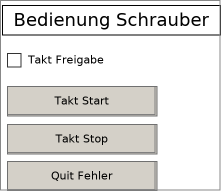
VISUALIZATION Frame_Schrauber_Bedien  // 221x191
VAR_IN_OUT
	bTaktFreigabe	:BOOL;
	bTaktStart		:BOOL;
	bTaktStop		:BOOL;
	bQuitError		:BOOL;
	
END_VAR
    Button (7,124 150x30), "Takt Stop"
        tap bTaktStop
    Button (7,86 150x30), "Takt Start"
        tap bTaktStart
    Checkbox (5,45 150x30), "Takt Freigabe", variable: bTaktFreigabe
    Rectangle (2,5 219x30), "Bedienung Schrauber"
    Button (7,161 150x30), "Quit Fehler"
        tap bQuitError
END_VISUALIZATION

(* stored: Version 1.1.0.1, ProductVersion 3.1.4024.15
   Visu Frame_Schrauber_Bedien: Id {208ad3ae-0579-4629-b70f-9aa68e5c0538} *)
